PROGRAM MAIN
VAR
  nTest : INT := 0;
END_VAR

nTest := nTest + 1;

TEST();

END_PROGRAM

(* stored: Version 1.1.0.1, ProductVersion 3.1.4024.10
   POU MAIN: Id {6c95b5c6-fc89-4a2a-a0f3-ac964d956dff}, SpecialFunc None *)
